# EPICS substitutions: ek9000App/Db/EL3312.substitutions
file EL3312.template
{       pattern
        {
                TERMINAL,

        }
        {
        }
}
